INTERFACE I_Sequence EXTENDS I_Object

METHOD PUBLIC M_Await 
VAR_INPUT
	Message:				STRING(255);
	tTimeout:				TIME;
	bCondition:				BOOL;
	nNumber:				INT;	
END_VAR
END_METHOD

END_INTERFACE

(* stored: Version 1.1.0.1
   Itf I_Sequence: Id {ab5e2af8-509e-42fb-9956-7609633302ce}
   Method M_Await: Id {e833a426-ec07-456c-8ba3-4d13a00bf184} *)
